% RSLogix 500 project I2A-JOB 22-MITCH_BAK149.RSS, saved by version 10.00.00.00 %
PROJECT "ML01B"    % processor: Bul.1763 MicroLogix 1100 Series B %

PROGRAM FILES
  LAD 2   8 rungs

DATA FILES
  O0 OUTPUT  4 elements
  I1 INPUT  6 elements
  S2 STATUS  66 elements
  B3 BINARY  1 elements
  T4 TIMER  1 elements
  C5 COUNTER  1 elements
  R6 CONTROL  1 elements
  N7 INTEGER  1 elements
  F8 FLOAT  1 elements

LADDER 2
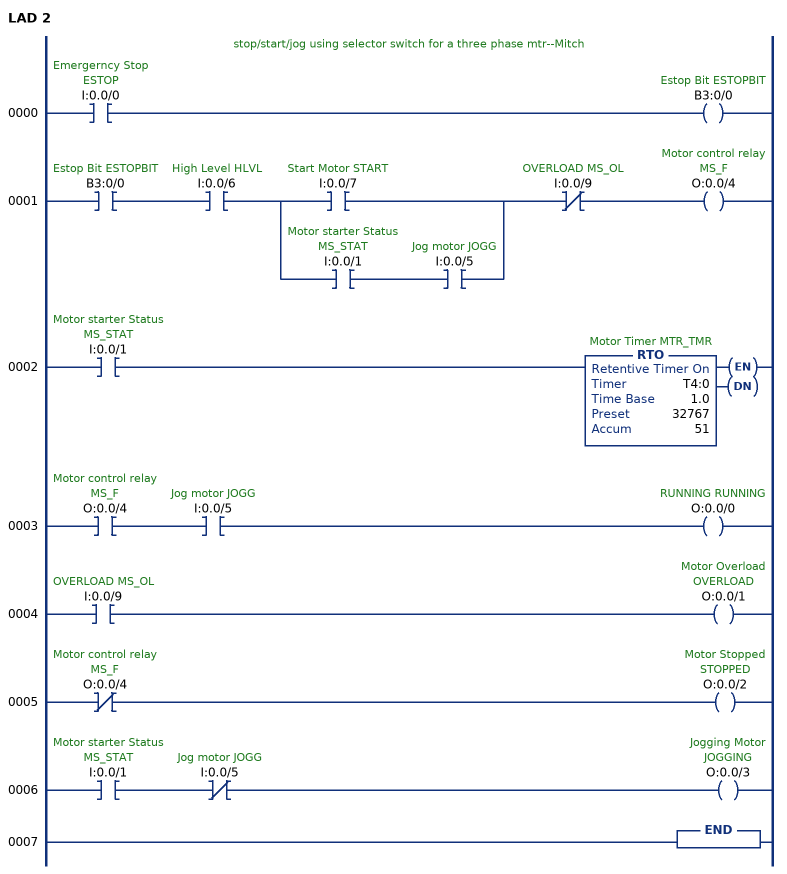
% Rung: 0 %
% stop/start/jog using selector switch for a three phase mtr--Mitch %
SOR XIC I:0.0/0 OTE B3:0/0 EOR
%   I:0.0/0  ESTOP  "Emergerncy Stop" %
%   B3:0/0  ESTOPBIT  "Estop Bit" %
% Rung: 1 %
SOR XIC B3:0/0 XIC I:0.0/6 BST XIC I:0.0/7 NXB XIC I:0.0/1 XIC I:0.0/5 BND XIO I:0.0/9 OTE O:0.0/4 EOR
%   B3:0/0  ESTOPBIT  "Estop Bit" %
%   I:0.0/6  HLVL  "High Level" %
%   I:0.0/7  START  "Start Motor" %
%   I:0.0/1  MS_STAT  "Motor starter Status" %
%   I:0.0/5  JOGG  "Jog motor" %
%   I:0.0/9  MS_OL  "OVERLOAD" %
%   O:0.0/4  MS_F  "Motor control relay" %
% Rung: 2 %
SOR XIC I:0.0/1 RTO T4:0 1.0 32767 51 EOR
%   I:0.0/1  MS_STAT  "Motor starter Status" %
%   T4:0  MTR_TMR  "Motor Timer" %
% Rung: 3 %
SOR XIC O:0.0/4 XIC I:0.0/5 OTE O:0.0/0 EOR
%   O:0.0/4  MS_F  "Motor control relay" %
%   I:0.0/5  JOGG  "Jog motor" %
%   O:0.0/0  RUNNING  "RUNNING" %
% Rung: 4 %
SOR XIC I:0.0/9 OTE O:0.0/1 EOR
%   I:0.0/9  MS_OL  "OVERLOAD" %
%   O:0.0/1  OVERLOAD  "Motor Overload" %
% Rung: 5 %
SOR XIO O:0.0/4 OTE O:0.0/2 EOR
%   O:0.0/4  MS_F  "Motor control relay" %
%   O:0.0/2  STOPPED  "Motor Stopped" %
% Rung: 6 %
SOR XIC I:0.0/1 XIO I:0.0/5 OTE O:0.0/3 EOR
%   I:0.0/1  MS_STAT  "Motor starter Status" %
%   I:0.0/5  JOGG  "Jog motor" %
%   O:0.0/3  JOGGING  "Jogging Motor" %
% Rung: 7 %
SOR END EOR

OTHER DOCUMENTED ADDRESSES
  B3:0/1  FWDB  "FWD BIT"
  B3:0/2  REVBIT  "REV BIT"
  B3:0/3  LAST_FWD  "LAST Forward"
  B3:0/4  LAST_REV  "Last Reverse"
  B3:0/5  RUN  "RUn Bit"
  B3:0/6  FJOG  "FWD Jog"
  B3:0/7  RJOG  "Rev Jog"
  B3:0/8  LATCH1  "LATCH"
  B3:0/9  UNLATCH  "Unlatch"
  I:0.0/2  MDR_STAT  "Motor Direction Contacts"
  I:0.0/3  AUTO__  "Mode on/off/auto"
  I:0.0/4  RUN__  "Mode on/auto/off"
  I:0.0/8  PB2  "Jog Motor"
  O:0.0/5  CR2ST  "Control relay 2"
  T4:0/DN  T4
  T4:0/TT  TTT
  T4:1/TT  TT

DATA TABLE (non-zero values as saved)
DATA B3
% B3:0 % 0X0101
DATA T4
% .PRE .ACC %
% T4:0 % 32767 51
DATA C5
% .PRE .ACC %
% C5:0 % 16 0
